// TIA Portal V18 export
// export: Created 2025-12-01T12:38:48.8884752Z, ExportSetting None, DisplayName Totally Integrated Automation Portal, DisplayVersion V18 Update 5, DisplayName TIA Portal Openness, DisplayVersion V18 Update 5, DisplayName TIA Portal Teamcenter Gateway, DisplayVersion V18, DisplayName TIA Portal Version Control Interface, DisplayVersion V18, DisplayName STEP 7 Professional, DisplayVersion V18 Update 5, DisplayName STEP 7 Safety, DisplayVersion V18, DisplayName WinCC Professional, DisplayVersion V18 Update 5
DATA_BLOCK "ST10_PLC_PutDB"   // DB902
{ S7_Optimized_Access := 'FALSE' }
// stored: AutoNumber false
   VAR
      OutData : Struct
         Global : Struct
            Beat : Bool;
            AutoRunning : Bool;
            Alarm : Bool;
            Spare_1 : Bool;
            Spare_2 : Bool;
            Spare_3 : Bool;
            Spare_4 : Bool;
            Spare_5 : Bool;
            Spare_6 : Bool;
            Spare_7 : Bool;
            Spare_8 : Bool;
            Spare_9 : Bool;
            Spare_10 : Bool;
            Spare_11 : Bool;
            Spare_12 : Bool;
            Spare_13 : Bool;
         END_STRUCT;
         Control : Struct
            PalletOut : Bool;
            Spare_16 : Bool;
            Spare_1 : Bool;
            Spare_2 : Bool;
            Spare_3 : Bool;
            Spare_4 : Bool;
            Spare_5 : Bool;
            Spare_6 : Bool;
            Spare_7 : Bool;
            Spare_8 : Bool;
            Spare_9 : Bool;
            Spare_10 : Bool;
            Spare_11 : Bool;
            Spare_12 : Bool;
            Spare_13 : Bool;
            Spare_14 : Byte;
            Spare_15 : Byte;
         END_STRUCT;
         Data : Struct
            Spare_5 : Int;
            Spare_4 : Int;
            Spare_1 : Int;
            Spare_2 : Int;
            Spare_6 : Int;   // Min
            Spare_3 : Array[0..83] of Byte;
         END_STRUCT;
      END_STRUCT;
   END_VAR
BEGIN
END_DATA_BLOCK
